// TIA Portal V17 export
// export: Created 2025-06-25T13:13:30.1485542Z, ExportSetting WithDefaults, DisplayName Totally Integrated Automation Portal, DisplayVersion V17 Update 8, DisplayName TIA Portal Openness, DisplayVersion V17 Update 8, DisplayName TIA Portal Version Control Interface, DisplayVersion V17, DisplayName STEP 7 Professional, DisplayVersion V17 Update 8, DisplayName STEP 7 Safety, DisplayVersion V17 Update 6, DisplayName WinCC Advanced, DisplayVersion V17 Update 8
TYPE "stPI_Regulator"
// stored: IsFailsafeCompliant false
   STRUCT
      bEnable : Bool;   // 1 = regulator on, 0 = regulator off
      fPV : Real;   // Process value
      fSP : Real;   // Setpoint
      fOutMax : Real;
      fOutMin : Real;
      fOut : Real;   // Manipulated value
      bManualMode : Bool;   // 1 = manual mode, 0 = auto
      fManualValue : Real;
      Kp : Real;   // Proportional gain
      Tn : Real;   // Integral gain (reset time)
      bAtMin : Bool;   // Controller negative saturation
      bAtMax : Bool;   // Controller positive saturation
      bFault : Bool;   // 1 = controller fault, 0 = ok
      nMode : USInt;   // 0 = Off, 1 = Auto, 2 = Manual
   END_STRUCT;
END_TYPE
